// TIA Portal V19 export
ORGANIZATION_BLOCK "Drives"   // OB1, FBD, ProgramCycle
TITLE = "Main Program Sweep (Cycle)"
{ S7_Optimized_Access := 'TRUE' }
// stored: SetENOAutomatically false
   VAR_INPUT
      Initial_Call : Bool;   // Initial call of this OB
      Remanence : Bool;   // =True, if remanent data are available
   END_VAR
BEGIN

REGION Network 1: 2510!
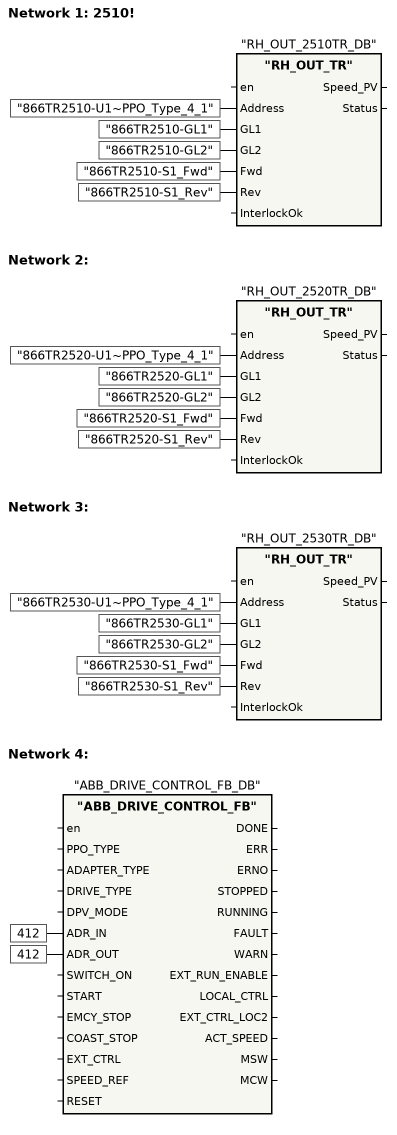
   "RH_OUT_2510TR_DB"(Address := "866TR2510-U1~PPO_Type_4_1",   // "RH_OUT_TR"
                      GL1 := "866TR2510-GL1",
                      GL2 := "866TR2510-GL2",
                      Fwd := "866TR2510-S1_Fwd",
                      Rev := "866TR2510-S1_Rev");
END_REGION

REGION Network 2
   "RH_OUT_2520TR_DB"(Address := "866TR2520-U1~PPO_Type_4_1",   // "RH_OUT_TR"
                      GL1 := "866TR2520-GL1",
                      GL2 := "866TR2520-GL2",
                      Fwd := "866TR2520-S1_Fwd",
                      Rev := "866TR2520-S1_Rev");
END_REGION

REGION Network 3
   "RH_OUT_2530TR_DB"(Address := "866TR2530-U1~PPO_Type_4_1",   // "RH_OUT_TR"
                      GL1 := "866TR2530-GL1",
                      GL2 := "866TR2530-GL2",
                      Fwd := "866TR2530-S1_Fwd",
                      Rev := "866TR2530-S1_Rev");
END_REGION

REGION Network 4
   "ABB_DRIVE_CONTROL_FB_DB"(ADR_IN := 412, ADR_OUT := 412);   // "ABB_DRIVE_CONTROL_FB"
END_REGION
END_ORGANIZATION_BLOCK
